SPLINE
SPL {X  -158.454, Y  +360.384, Z    +0.000, E1  +340.634, E3 -480540.576}
SPL {X  -159.737, Y  +373.507, Z    +0.000, E1  +349.689, E3 -480562.611}
SPL {X  -159.990, Y  +382.574, Z    +0.000, E1  +355.537, E3 -480569.299}
SPL {X  -159.990, Y  +389.909, Z    +0.000, E1  +360.662, E3 -480573.313}
SPL {X  -159.990, Y  +396.289, Z    +0.000, E1  +365.500, E3 -480577.093}
SPL {X  -159.990, Y  +407.941, Z    +0.000, E1  +374.126, E3 -480588.430}
SPL {X  -159.990, Y  +418.671, Z    +0.000, E1  +379.855, E3 -480607.847}
SPL {X  -159.990, Y  +429.878, Z    +0.000, E1  +383.330, E3 -480637.902}
SPL {X  -159.990, Y  +432.103, Z    +0.000, E1  +383.301, E3 -480648.920}
SPL {X  -159.990, Y  +434.188, Z    +0.000, E1  +383.325, E3 -480659.117}
SPL {X  -159.990, Y  +437.007, Z    +0.000, E1  +383.323, E3 -480673.008}
SPL {X  -159.990, Y  +439.778, Z    +0.000, E1  +383.323, E3 -480686.640}
SPL {X  -159.990, Y  +442.945, Z    +0.000, E1  +383.339, E3 -480702.204}
SPL {X  -159.990, Y  +446.037, Z    +0.000, E1  +383.324, E3 -480717.455}
SPL {X  -159.990, Y  +448.341, Z    +0.000, E1  +383.317, E3 -480728.772}
SPL {X  -159.990, Y  +450.345, Z    +0.000, E1  +383.316, E3 -480738.650}
SPL {X  -159.990, Y  +452.828, Z    +0.000, E1  +383.330, E3 -480750.849}
SPL {X  -159.990, Y  +456.338, Z    +0.000, E1  +383.359, E3 -480768.042}
SPL {X  -159.990, Y  +459.480, Z    +0.000, E1  +383.323, E3 -480783.583}
SPL {X  -159.990, Y  +462.520, Z    +0.000, E1  +383.350, E3 -480798.487}
SPL {X  -159.990, Y  +465.602, Z    +0.000, E1  +383.328, E3 -480813.687}
SPL {X  -159.990, Y  +467.934, Z    +0.000, E1  +383.321, E3 -480825.181}
SPL {X  -159.990, Y  +469.939, Z    +0.000, E1  +383.319, E3 -480835.043}
SPL {X  -159.990, Y  +472.144, Z    +0.000, E1  +383.327, E3 -480845.894}
SPL {X  -159.990, Y  +474.152, Z    +0.000, E1  +383.309, E3 -480855.846}
SPL {X  -159.990, Y  +476.560, Z    +0.000, E1  +383.332, E3 -480867.654}
SPL {X  -159.990, Y  +478.770, Z    +0.000, E1  +383.306, E3 -480878.579}
SPL {X  -159.990, Y  +480.905, Z    +0.000, E1  +383.327, E3 -480889.047}
SPL {X  -159.990, Y  +484.251, Z    +0.000, E1  +383.352, E3 -480905.463}
SPL {X  -159.990, Y  +488.031, Z    +0.000, E1  +383.345, E3 -480924.096}
SPL {X  -159.990, Y  +491.121, Z    +0.000, E1  +383.323, E3 -480939.341}
SPL {X  -159.990, Y  +493.610, Z    +0.000, E1  +383.323, E3 -480951.594}
SPL {X  -159.990, Y  +496.863, Z    +0.000, E1  +383.350, E3 -480967.554}
SPL {X  -159.990, Y  +499.995, Z    +0.000, E1  +383.324, E3 -480983.015}
SPL {X  -159.990, Y  +502.341, Z    +0.000, E1  +383.320, E3 -480994.574}
SPL {X  -159.990, Y  +505.377, Z    +0.000, E1  +383.346, E3 -481009.465}
SPL {X  -159.990, Y  +508.024, Z    +0.000, E1  +383.315, E3 -481022.547}
SPL {X  -159.990, Y  +510.344, Z    +0.000, E1  +383.327, E3 -481033.954}
SPL {X  -159.990, Y  +513.289, Z    +0.000, E1  +383.332, E3 -481048.444}
SPL {X  -159.990, Y  +516.195, Z    +0.000, E1  +383.325, E3 -481062.763}
SPL {X  -159.990, Y  +518.925, Z    +0.000, E1  +383.333, E3 -481076.126}
SPL {X  -159.990, Y  +521.408, Z    +0.000, E1  +383.329, E3 -481088.335}
SPL {X  -159.990, Y  +523.942, Z    +0.000, E1  +383.333, E3 -481100.828}
SPL {X  -159.990, Y  +527.007, Z    +0.000, E1  +383.339, E3 -481115.928}
SPL {X  -159.990, Y  +529.993, Z    +0.000, E1  +383.329, E3 -481130.630}
SPL {X  -159.990, Y  +532.441, Z    +0.000, E1  +383.322, E3 -481142.681}
SPL {X  -159.990, Y  +534.618, Z    +0.000, E1  +383.322, E3 -481153.414}
SPL {X  -159.990, Y  +537.024, Z    +0.000, E1  +383.321, E3 -481165.276}
SPL {X  -159.990, Y  +539.129, Z    +0.000, E1  +383.310, E3 -481175.659}
SPL {X  -159.990, Y  +541.183, Z    +0.000, E1  +383.319, E3 -481185.756}
SPL {X  -159.990, Y  +543.647, Z    +0.000, E1  +383.325, E3 -481197.859}
SPL {X  -159.990, Y  +545.957, Z    +0.000, E1  +383.318, E3 -481209.239}
SPL {X  -159.990, Y  +548.912, Z    +0.000, E1  +383.354, E3 -481223.699}
SPL {X  -159.990, Y  +551.655, Z    +0.000, E1  +383.320, E3 -481237.274}
SPL {X  -159.990, Y  +553.711, Z    +0.000, E1  +383.317, E3 -481247.396}
SPL {X  -159.990, Y  +555.637, Z    +0.000, E1  +383.323, E3 -481256.864}
SPL {X  -159.990, Y  +558.758, Z    +0.000, E1  +383.351, E3 -481272.174}
SPL {X  -159.990, Y  +561.830, Z    +0.000, E1  +383.325, E3 -481287.347}
SPL {X  -159.990, Y  +564.273, Z    +0.000, E1  +383.325, E3 -481299.372}
SPL {X  -159.990, Y  +567.351, Z    +0.000, E1  +383.348, E3 -481314.467}
SPL {X  -159.990, Y  +570.314, Z    +0.000, E1  +383.326, E3 -481329.099}
SPL {X  -159.990, Y  +572.504, Z    +0.000, E1  +383.321, E3 -481339.884}
SPL {X  -159.990, Y  +575.653, Z    +0.000, E1  +383.355, E3 -481355.321}
SPL {X  -159.990, Y  +578.932, Z    +0.000, E1  +383.330, E3 -481371.504}
SPL {X  -159.990, Y  +581.497, Z    +0.000, E1  +383.329, E3 -481384.088}
SPL {X  -159.990, Y  +583.973, Z    +0.000, E1  +383.332, E3 -481396.274}
SPL {X  -159.990, Y  +586.020, Z    +0.000, E1  +383.323, E3 -481406.357}
SPL {X  -159.990, Y  +587.711, Z    +0.000, E1  +383.318, E3 -481414.697}
SPL {X  -159.990, Y  +589.763, Z    +0.000, E1  +383.328, E3 -481424.773}
SPL {X  -159.990, Y  +591.698, Z    +0.000, E1  +383.324, E3 -481434.258}
SPL {X  -159.990, Y  +593.847, Z    +0.000, E1  +383.340, E3 -481444.789}
SPL {X  -159.990, Y  +597.018, Z    +0.000, E1  +383.367, E3 -481460.321}
SPL {X  -159.990, Y  +599.887, Z    +0.000, E1  +383.341, E3 -481474.425}
SPL {X  -159.990, Y  +601.949, Z    +0.000, E1  +383.344, E3 -481484.552}
SPL {X  -159.990, Y  +605.106, Z    +0.000, E1  +383.383, E3 -481499.998}
SPL {X  -159.990, Y  +608.111, Z    +0.000, E1  +383.342, E3 -481514.849}
SPL {X  -159.990, Y  +610.073, Z    +0.000, E1  +383.343, E3 -481524.507}
SPL {X  -159.990, Y  +613.021, Z    +0.000, E1  +383.365, E3 -481538.977}
SPL {X  -159.990, Y  +615.657, Z    +0.000, E1  +383.331, E3 -481552.025}
SPL {X  -159.990, Y  +617.658, Z    +0.000, E1  +383.335, E3 -481561.867}
SPL {X  -159.990, Y  +620.788, Z    +0.000, E1  +383.368, E3 -481577.201}
SPL {X  -159.990, Y  +624.347, Z    +0.000, E1  +383.355, E3 -481594.721}
SPL {X  -159.990, Y  +627.144, Z    +0.000, E1  +383.340, E3 -481608.490}
SPL {X  -159.990, Y  +629.284, Z    +0.000, E1  +383.339, E3 -481618.998}
SPL {X  -159.990, Y  +631.206, Z    +0.000, E1  +383.337, E3 -481628.452}
SPL {X  -159.990, Y  +633.318, Z    +0.000, E1  +383.339, E3 -481638.857}
SPL {X  -159.990, Y  +635.650, Z    +0.000, E1  +383.339, E3 -481650.327}
SPL {X  -159.990, Y  +637.597, Z    +0.000, E1  +383.330, E3 -481659.950}
SPL {X  -159.990, Y  +640.369, Z    +0.000, E1  +383.354, E3 -481673.584}
SPL {X  -159.990, Y  +644.241, Z    +0.000, E1  +383.355, E3 -481692.696}
SPL {X  -159.990, Y  +648.287, Z    +0.000, E1  +383.349, E3 -481712.653}
SPL {X  -159.990, Y  +651.427, Z    +0.000, E1  +383.319, E3 -481728.148}
SPL {X  -159.990, Y  +653.536, Z    +0.000, E1  +383.313, E3 -481738.530}
SPL {X  -159.990, Y  +656.380, Z    +0.000, E1  +383.347, E3 -481752.465}
SPL {X  -159.990, Y  +659.180, Z    +0.000, E1  +383.314, E3 -481766.314}
SPL {X  -159.990, Y  +661.392, Z    +0.000, E1  +383.318, E3 -481777.207}
SPL {X  -159.990, Y  +663.662, Z    +0.000, E1  +383.322, E3 -481788.331}
SPL {X  -159.990, Y  +665.964, Z    +0.000, E1  +383.328, E3 -481799.622}
SPL {X  -159.990, Y  +667.870, Z    +0.000, E1  +383.320, E3 -481809.029}
SPL {X  -159.990, Y  +669.861, Z    +0.000, E1  +383.321, E3 -481818.830}
SPL {X  -159.990, Y  +671.893, Z    +0.000, E1  +383.319, E3 -481828.838}
SPL {X  -159.974, Y  +673.789, Z    +0.000, E1  +383.323, E3 -481838.154}
SPL {X  -159.924, Y  +676.110, Z    +0.000, E1  +383.320, E3 -481849.638}
SPL {X  -159.801, Y  +679.265, Z    +0.000, E1  +383.327, E3 -481865.257}
SPL {X  -159.626, Y  +682.287, Z    +0.000, E1  +383.280, E3 -481880.355}
SPL {X  -159.462, Y  +684.486, Z    +0.000, E1  +383.258, E3 -481891.355}
SPL {X  -159.289, Y  +686.457, Z    +0.000, E1  +383.223, E3 -481901.265}
SPL {X  -159.052, Y  +688.801, Z    +0.000, E1  +383.217, E3 -481913.000}
SPL {X  -158.770, Y  +691.222, Z    +0.000, E1  +383.158, E3 -481925.258}
SPL {X  -158.553, Y  +692.896, Z    +0.000, E1  +383.130, E3 -481933.723}
ENDSPLINE

SPLINE
SPL {X  -159.063, Y  +688.696, Z    +0.000, E1  +377.094, E3 -481971.844}
SPL {X  -159.987, Y  +672.488, Z    +0.000, E1  +365.638, E3 -481995.909}
SPL {X  -159.990, Y  +663.928, Z    +0.000, E1  +359.662, E3 -482001.703}
SPL {X  -159.990, Y  +658.009, Z    +0.000, E1  +355.226, E3 -482005.403}
SPL {X  -159.990, Y  +651.879, Z    +0.000, E1  +350.548, E3 -482010.466}
SPL {X  -159.990, Y  +637.832, Z    +0.000, E1  +341.694, E3 -482028.057}
SPL {X  -159.990, Y  +626.634, Z    +0.000, E1  +337.968, E3 -482058.910}
SPL {X  -159.990, Y  +624.622, Z    +0.000, E1  +337.980, E3 -482069.493}
SPL {X  -159.990, Y  +622.489, Z    +0.000, E1  +337.969, E3 -482080.660}
SPL {X  -159.990, Y  +619.267, Z    +0.000, E1  +337.938, E3 -482097.494}
SPL {X  -159.990, Y  +615.467, Z    +0.000, E1  +337.940, E3 -482117.430}
SPL {X  -159.990, Y  +612.600, Z    +0.000, E1  +337.975, E3 -482132.541}
SPL {X  -159.990, Y  +610.646, Z    +0.000, E1  +337.979, E3 -482142.798}
SPL {X  -159.990, Y  +608.810, Z    +0.000, E1  +337.977, E3 -482152.431}
SPL {X  -159.990, Y  +605.804, Z    +0.000, E1  +337.936, E3 -482168.076}
SPL {X  -159.990, Y  +602.819, Z    +0.000, E1  +337.963, E3 -482183.748}
SPL {X  -159.990, Y  +600.642, Z    +0.000, E1  +337.968, E3 -482195.176}
SPL {X  -159.990, Y  +598.568, Z    +0.000, E1  +337.954, E3 -482205.969}
SPL {X  -159.990, Y  +596.440, Z    +0.000, E1  +337.964, E3 -482217.150}
SPL {X  -159.990, Y  +593.768, Z    +0.000, E1  +337.929, E3 -482231.083}
SPL {X  -159.990, Y  +590.068, Z    +0.000, E1  +337.924, E3 -482250.451}
SPL {X  -159.990, Y  +586.620, Z    +0.000, E1  +337.935, E3 -482268.514}
SPL {X  -159.990, Y  +584.080, Z    +0.000, E1  +337.953, E3 -482281.840}
SPL {X  -159.990, Y  +581.924, Z    +0.000, E1  +337.949, E3 -482293.141}
SPL {X  -159.990, Y  +579.673, Z    +0.000, E1  +337.950, E3 -482304.939}
SPL {X  -159.990, Y  +576.961, Z    +0.000, E1  +337.936, E3 -482319.118}
SPL {X  -159.990, Y  +574.188, Z    +0.000, E1  +337.947, E3 -482333.665}
SPL {X  -159.990, Y  +571.954, Z    +0.000, E1  +337.959, E3 -482345.423}
SPL {X  -159.990, Y  +570.110, Z    +0.000, E1  +337.958, E3 -482355.073}
SPL {X  -159.990, Y  +568.165, Z    +0.000, E1  +337.957, E3 -482365.253}
SPL {X  -159.990, Y  +565.292, Z    +0.000, E1  +337.922, E3 -482380.231}
SPL {X  -159.990, Y  +562.598, Z    +0.000, E1  +337.958, E3 -482394.443}
SPL {X  -159.990, Y  +560.652, Z    +0.000, E1  +337.962, E3 -482404.654}
SPL {X  -159.990, Y  +558.143, Z    +0.000, E1  +337.928, E3 -482417.686}
SPL {X  -159.990, Y  +555.329, Z    +0.000, E1  +337.943, E3 -482432.430}
SPL {X  -159.990, Y  +553.115, Z    +0.000, E1  +337.946, E3 -482444.036}
SPL {X  -159.990, Y  +550.886, Z    +0.000, E1  +337.944, E3 -482455.717}
SPL {X  -159.990, Y  +548.568, Z    +0.000, E1  +337.944, E3 -482467.838}
SPL {X  -159.990, Y  +546.537, Z    +0.000, E1  +337.948, E3 -482478.473}
SPL {X  -159.990, Y  +545.062, Z    +0.000, E1  +337.955, E3 -482486.232}
SPL {X  -159.990, Y  +543.060, Z    +0.000, E1  +337.943, E3 -482496.711}
SPL {X  -159.990, Y  +539.928, Z    +0.000, E1  +337.917, E3 -482513.052}
SPL {X  -159.990, Y  +536.935, Z    +0.000, E1  +337.942, E3 -482528.769}
SPL {X  -159.990, Y  +534.656, Z    +0.000, E1  +337.946, E3 -482540.713}
SPL {X  -159.990, Y  +532.453, Z    +0.000, E1  +337.944, E3 -482552.240}
SPL {X  -159.990, Y  +530.660, Z    +0.000, E1  +337.952, E3 -482561.643}
SPL {X  -159.990, Y  +528.702, Z    +0.000, E1  +337.939, E3 -482571.856}
SPL {X  -159.990, Y  +525.760, Z    +0.000, E1  +337.914, E3 -482587.197}
SPL {X  -159.990, Y  +522.838, Z    +0.000, E1  +337.933, E3 -482602.564}
SPL {X  -159.990, Y  +519.698, Z    +0.000, E1  +337.916, E3 -482618.947}
SPL {X  -159.990, Y  +517.251, Z    +0.000, E1  +337.946, E3 -482631.807}
SPL {X  -159.990, Y  +515.568, Z    +0.000, E1  +338.084, E3 -482641.904}
ENDSPLINE

SPLINE
SPL {X  -159.990, Y  +517.293, Z    +0.000, E1  +340.923, E3 -482658.202}
ENDSPLINE

SPLINE
SPL {X  -159.990, Y  +512.548, Z    +0.000, E1  +339.587, E3 -482673.777}
SPL {X  -159.990, Y  +508.660, Z    +0.000, E1  +338.515, E3 -482685.831}
SPL {X  -159.990, Y  +503.499, Z    +0.000, E1  +337.116, E3 -482700.911}
SPL {X  -159.990, Y  +498.406, Z    +0.000, E1  +335.789, E3 -482714.944}
SPL {X  -159.990, Y  +494.630, Z    +0.000, E1  +334.924, E3 -482725.666}
ENDSPLINE

SLIN {X  -200.000, Y  +530.000, E1    +0.000}
HALT
END
